// TIA Portal V16 export
// export: Created 2021-04-11T09:51:29.5049016Z, ExportSetting WithDefaults, DisplayName Totally Integrated Automation Portal, DisplayVersion V16, DisplayName TIA Portal Version Control Interface, DisplayVersion V16, DisplayName TIA Portal Openness, DisplayVersion V16, DisplayName STEP 7 Professional, DisplayVersion V16, DisplayName STEP 7 Safety, DisplayVersion V16, DisplayName WinCC Unified SCADA Engineering System, DisplayVersion V16
TYPE "dateTime"
// stored: IsFailsafeCompliant false
   STRUCT
      year : Int;
      month : Int;
      day : Int;
      hour : Int;
      minute : Int;
      second : Int;
   END_STRUCT;
END_TYPE
